# B&R Automation Studio project A2019059_Linka_Power_CP (part 62)

#### Main.st - Init, cyclic, exit code
```iecst
// ----------------------------------------------------------------------------------------
//	Function:	mappView explorer
//  Version:	1.00
//	Changed:	07.01.2020
// ----------------------------------------------------------------------------------------

PROGRAM _INIT
	// ----------------------------------------------------------------------------------------
	// Copy pre-configured devices into list
	brsmemcpy(ADR(EXPL.PAR[0].device_list), ADR(EXPL_DEVICE_LIST), SIZEOF(EXPL_DEVICE_LIST));
	brsmemcpy(ADR(EXPL.PAR[1].device_list), ADR(EXPL_DEVICE_LIST), SIZEOF(EXPL_DEVICE_LIST));
	brsstrcpy(ADR(EXPL.PAR[0].device_active), ADR(EXPL.PAR[0].device_list[0]));
	brsstrcpy(ADR(EXPL.PAR[1].device_active), ADR(EXPL.PAR[1].device_list[0]));

	// ----------------------------------------------------------------------------------------
	// Allocate memory for file upload and download
	AsMemPartCreate_0.enable	:= TRUE;
	AsMemPartCreate_0.len		:= EXPL_UPLOAD_DOWNLOAD_SIZE;
	AsMemPartCreate_0();
	IF AsMemPartCreate_0.status <> 0 THEN
		step := CreateError(ERR_MEM_ALLOC, side, step, 'file upload and download alloc failed', ADR(EXPL));
	ELSE
		AsMemPartAllocClear_0.enable	:= TRUE;
		AsMemPartAllocClear_0.ident		:= AsMemPartCreate_0.ident;
		AsMemPartAllocClear_0.len		:= EXPL_UPLOAD_DOWNLOAD_SIZE;
		AsMemPartAllocClear_0();
		IF AsMemPartCreate_0.status <> 0 THEN
			step := CreateError(ERR_MEM_ALLOC, side, step, 'file upload and download clear failed', ADR(EXPL));
		END_IF
	END_IF

	// ----------------------------------------------------------------------------------------
	// Generate HTML messages for web upload
	upload_response[0]	:= '<html><body><form action="/uploadA.html" name="form_upload" method="post" enctype="multipart/form-data" >
	<label for="file-upload" style="font-weight:bold;font-family: sans-serif;font-size:16px;padding:10px 10px;10px;10px;" class="custom-file-upload">Upload</label>
	<input type="file" id="file-upload" style="display:none;" onchange="form.submit()" name="file_selected" content-type="application/octet-stream" />
	</form><body></html> ';
	WebServiceUpload[0].pServiceName := ADR('uploadA.html');
	upload_response[1]	:= '<html><body><form action="/uploadB.html" name="form_upload" method="post" enctype="multipart/form-data" >
	<label for="file-upload" style="font-weight:bold;font-family: sans-serif;font-size:16px;padding:10px 10px;10px;10px;" class="custom-file-upload">Upload</label>
	<input type="file" id="file-upload" style="display:none;" onchange="form.submit()" name="file_selected" content-type="application/octet-stream" />
	</form><body></html> ';
	WebServiceUpload[1].pServiceName := ADR('uploadB.html');
END_PROGRAM

PROGRAM _CYCLIC
	// ----------------------------------------------------------------------------------------
	// Web service driver for file upload
	WebServiceUpload[side].enable 			:= TRUE;
	WebServiceUpload[side].option 			:= httpOPTION_HTTP_11 + httpOPTION_SERVICE_TYPE_NAME;
	WebServiceUpload[side].pRequestData  	:= AsMemPartAllocClear_0.mem;
	WebServiceUpload[side].requestDataSize 	:= EXPL_UPLOAD_DOWNLOAD_SIZE;
	WebServiceUpload[side].pResponseData 	:= ADR(upload_response[side]);
	WebServiceUpload[side].responseDataLen 	:= brsstrlen(ADR(upload_response[side]));
	WebServiceUpload[side]();

	// Reset send command
	IF(WebServiceUpload[side].send = TRUE)  THEN
		WebServiceUpload[side].send := FALSE;
	// Send response when page is loaded or data is posted
	ELSIF(WebServiceUpload[side].status = ERR_OK AND WebServiceUpload[side].send = FALSE) THEN
		WebServiceUpload[side].send := TRUE;
	// New upload data arrived
	ELSIF(WebServiceUpload[side].send = FALSE AND WebServiceUpload[side].requestDataLen > 0) THEN
		EXPL.CMD[side].upload := 1;
	END_IF

	// ------------------------------------------------------------------------------------------------
	// Set switches for HMI, these buttons are enabled if there is at least one file or directory
	IF(EXPL.DAT[side].item_num > 0) THEN
		EXPL.VIS[side].enable_button_set_1 := 1;
	ELSE
		EXPL.VIS[side].enable_button_set_1 := 0;
	END_IF

	// ------------------------------------------------------------------------------------------------
	// Generate device name list for drop down box
	brsmemset(ADR(EXPL.VIS[side].device_list), 0, SIZEOF(EXPL.VIS[side].device_list));
	FOR lx := 0 TO SIZEOF(EXPL.VIS[side].device_list)/SIZEOF(EXPL.VIS[side].device_list[0]) - 1 DO
		IF (EXPL.PAR[side].device_list[lx] <> '') THEN
			String2DataProvider(ADR(EXPL.PAR[side].device_list[lx]), ADR(EXPL.VIS[side].device_list[lx]));
		END_IF
	END_FOR;

	// ------------------------------------------------------------------------------------------------
	// Handle double click for directory change and file view
	IF(EXPL.VIS[side].double_click_event > 0) THEN
		double_click_timer.PT := 50;
		double_click_timer.IN := 1;
		double_click_timer();
		IF(EXPL.VIS[side].double_click_event > 1) THEN
			double_click_timer.IN := 0;
			double_click_timer();
			EXPL.VIS[side].double_click_event := 0;
			IF(brsmemcmp(ADR(EXPL.DAT[side].item_list[EXPL.VIS[side].item_selected]), ADR('(DIR)'), 5) = 0 OR EXPL.DAT[side].item_list[EXPL.VIS[side].item_selected] = '..') THEN
				EXPL.CMD[side].dir_change := 1;
			ELSE
				EXPL.CMD[side].view_file := 1;
			END_IF
		END_IF
	END_IF
	IF(double_click_timer.Q) THEN
		double_click_timer.IN := 0;
		double_click_timer();
		IF(EXPL.VIS[side].double_click_event > 0) THEN
			EXPL.VIS[side].double_click_event := EXPL.VIS[side].double_click_event - 1;
		END_IF
	END_IF

	//--------------------------------------------------------------------------------------------------
	// Check if parameters are valid
	IF (EXPL.PAR[side].device_active = '') THEN
		step := CreateError(ERR_DEVICE_UNDEFINED, side, step, 'device is not defined', ADR(EXPL));
		RETURN;
	END_IF
	IF (brsstrlen(ADR(EXPL.PAR[side].dir_path)) >= EXPL_DIR_PATH_LENGTH) THEN
		step := CreateError(ERR_PATH_CRITICAL, side, step, 'directory path critical error', ADR(EXPL));
		RETURN;
	END_IF

	// ------------------------------------------------------------------------------------------------
	// Track filter change
	IF (FILTER_AUTO_REFRESH AND brsstrcmp(ADR(old_filter[side]), ADR(EXPL.PAR[side].item_filter)) <> 0) THEN
		brsstrcpy(ADR(old_filter[side]), ADR(EXPL.PAR[side].item_filter));
		EXPL.CMD[side].refresh	:= 1;
	END_IF

	// ------------------------------------------------------------------------------------------------
	// Track device name change
	IF(device_active_old[side] <> EXPL.PAR[side].device_active) THEN
		EXPL.PAR[side].dir_path := '';
		EXPL.CMD[side].refresh	:= 1;
	END_IF
	device_active_old[side] := EXPL.PAR[side].device_active;

	// ------------------------------------------------------------------------------------------------
	// Stop here if no command is set
	IF (EXPL.CMD[side].refresh = 0 AND EXPL.CMD[side].dir_change = 0 AND EXPL.CMD[side].dir_create = 0 AND EXPL.CMD[side].copy = 0 AND EXPL.CMD[side].copy_all = 0 AND EXPL.CMD[side].delete = 0 AND EXPL.CMD[side].rename = 0 AND EXPL.CMD[side].view_file = 0 AND EXPL.CMD[side].download = 0 AND EXPL.CMD[side].upload = 0) THEN
		// --------------------------------------------------------------------------------------------
		// Show current state
		EXPL.status := 'Waiting...';
		// --------------------------------------------------------------------------------------------
		// If selection is out of range set it to maximum
		IF ((EXPL.VIS[side].item_selected > EXPL.DAT[side].item_num - 1) AND (EXPL.DAT[side].item_num <> 0)) THEN
			EXPL.VIS[side].item_selected := EXPL.DAT[side].item_num - 1;
		END_IF
		side := NOT side;
		// Enable buttons when command is active
		EXPL.VIS[0].enable_button_set_2 := 1;
		EXPL.VIS[1].enable_button_set_2 := 1;
		RETURN;
	END_IF

	// Disable buttons when command is active
	EXPL.VIS[0].enable_button_set_1 := 0;
	EXPL.VIS[1].enable_button_set_1 := 0;
	EXPL.VIS[0].enable_button_set_2 := 0;
	EXPL.VIS[1].enable_button_set_2 := 0;
	//**************************************************************************************************
	// Cyclic Part
	//**************************************************************************************************
	CASE step OF
		//**********************************************************************************************
		// Wait for command
		//**********************************************************************************************
		EXP_WAIT:
			// ----------------------------------------------------------------------------------------
			// Refresh direcrory information
			IF (EXPL.CMD[side].refresh = 1) THEN
				step := EXP_READ_DIR;
			END_IF
			// ----------------------------------------------------------------------------------------
			// Change active directory
			IF (EXPL.CMD[side].dir_change = 1) THEN
				// ------------------------------------------------------------------------------------
				// Check if directory name is empty
				IF (EXPL.DAT[side].item_list[EXPL.VIS[side].item_selected] = '') THEN
				step := CreateError(ERR_EMPTY_ITEM, side, step, 'directory name is empty', ADR(EXPL));
				// Check if directory name is valid
				ELSIF((brsmemcmp(ADR(EXPL.DAT[side].item_list[EXPL.VIS[side].item_selected]), ADR('(DIR)'), 5) <> 0) AND (EXPL.DAT[side].item_list[EXPL.VIS[side].item_selected] <> '..'))  THEN
					step := CreateError(ERR_INVALID_ITEM_NAME, side, step, 'this is not a valid directory name', ADR(EXPL));
				// Check if new directory name fits into string
				ELSIF(brsstrlen(ADR(EXPL.DAT[side].item_list[EXPL.VIS[side].item_selected])) - 5 + brsstrlen(ADR(EXPL.PAR[side].dir_path)) + 1 >= EXPL_DIR_PATH_LENGTH) THEN
					step := CreateError(ERR_PATH_EXCEEDS_MAX, side, step, 'directory path exceeds maximum length', ADR(EXPL));
				ELSE
					step := EXP_DIR_CHANGE;
				END_IF
			END_IF
			// ----------------------------------------------------------------------------------------
			// Create a new directory
			IF (EXPL.CMD[side].dir_create = 1) THEN
				// ------------------------------------------------------------------------------------
				// Check if new directory name is empty
				IF (EXPL.PAR[side].new_name = '') THEN
					step := CreateError(ERR_EMPTY_ITEM, side, step, 'directory name is empty', ADR(EXPL));
				// Check if new directory name fits into path string
				ELSIF(brsstrlen(ADR(EXPL.PAR[side].new_name)) + brsstrlen(ADR(EXPL.PAR[side].dir_path)) + 1 >= EXPL_DIR_PATH_LENGTH) THEN
					step := CreateError(ERR_PATH_EXCEEDS_MAX, side, step, 'directory path name exceeds maximum length', ADR(EXPL));
				// Check if new directory name fits into directory name string
				ELSIF(brsstrlen(ADR(EXPL.PAR[side].new_name)) + 5 >= EXPL_ITEM_LENGTH) THEN
					step := CreateError(ERR_DIR_EXCEEDS_MAX, side, step, 'directory name exceeds maximum length', ADR(EXPL));
				ELSE
					step := EXP_DIR_CREATE;
				END_IF
			END_IF
			// ----------------------------------------------------------------------------------------
			// Copy one file
			IF (EXPL.CMD[side].copy = 1) THEN
				// ------------------------------------------------------------------------------------
				// Make sure that user chooses a valid item
				IF (EXPL.DAT[side].item_list[EXPL.VIS[side].item_selected] = '..') THEN
					step := CreateError(ERR_INVALID_ITEM_NAME, side, step, 'this is not a valid item name', ADR(EXPL));
				ELSIF(brsmemcmp(ADR(EXPL.DAT[side].item_list[EXPL.VIS[side].item_selected]), ADR('(DIR)'), 5) = 0)	THEN
					step := EXP_DIR_COPY;
				ELSE
					step := EXP_FILE_COPY;
				END_IF
			END_IF
			// ----------------------------------------------------------------------------------------
			// Copy all files and folders in this directory
			IF (EXPL.CMD[side].copy_all = 1) THEN
				step := EXP_COPY_ALL;
			END_IF
			// ----------------------------------------------------------------------------------------
			// View selected file
			IF (EXPL.CMD[side].view_file = 1) THEN
				step := EXP_FILE_VIEW;
			END_IF
			// ----------------------------------------------------------------------------------------
			// Download selected file
			IF (EXPL.CMD[side].download = 1) THEN
				// Make sure download is not directory
				IF(brsmemcmp(ADR(EXPL.DAT[side].item_list[EXPL.VIS[side].item_selected]), ADR('(DIR)'), 5) <> 0) THEN
					EXPL.VIS[side].download_file_url := '';
					step := EXP_FILE_DOWNLOAD;
				ELSE
					step := CreateError(ERR_DIR_DOWNLOAD, side, step, 'downloading a directory is not supported', ADR(EXPL));
				END_IF
			END_IF
			// ----------------------------------------------------------------------------------------
			// Upload a new file
			IF (EXPL.CMD[side].upload = 1) THEN
				step := EXP_FILE_UPLOAD;
			END_IF
			// ----------------------------------------------------------------------------------------
			// Delete the selected file
			IF (EXPL.CMD[side].delete = 1) THEN
				// Check if directory name is empty
				IF (EXPL.DAT[side].item_list[EXPL.VIS[side].item_selected] = '')	THEN
					step := CreateError(ERR_EMPTY_ITEM, side, step, 'item name is empty', ADR(EXPL));
				// Check if new directory name fits into string
				ELSIF(brsstrlen(ADR(EXPL.DAT[side].item_list[EXPL.VIS[side].item_selected])) + brsstrlen(ADR(EXPL.PAR[side].dir_path)) + 1 >= EXPL_DIR_PATH_LENGTH + EXPL_ITEM_LENGTH) THEN
					step := CreateError(ERR_PATH_EXCEEDS_MAX, side, step, 'directory path exceeds maximum length', ADR(EXPL));
				// Make sure that a valid item was selected
				ELSIF(EXPL.DAT[side].item_list[EXPL.VIS[side].item_selected] = '..') THEN
					step := CreateError(ERR_INVALID_ITEM_NAME, side, step, 'this is not a valid item name', ADR(EXPL));
				// Delete a directory
				ELSIF(brsmemcmp(ADR(EXPL.DAT[side].item_list[EXPL.VIS[side].item_selected]), ADR('(DIR)'), 5) = 0)	THEN
					step := EXP_DIR_DELETE;
				// Delete a file
				ELSE
					step := EXP_FILE_DELETE;
				END_IF
			END_IF
			// ----------------------------------------------------------------------------------------
			// Rename file or directory
			IF (EXPL.CMD[side].rename = 1) THEN
				// ------------------------------------------------------------------------------------
				// Check if new directory name is empty
				IF (EXPL.PAR[side].new_name = '') THEN
					step := CreateError(ERR_EMPTY_ITEM, side, step, 'new name is empty', ADR(EXPL));
				// Make sure that a valid item was selected
				ELSIF (EXPL.DAT[side].item_list[EXPL.VIS[side].item_selected] = '..') THEN
					step := CreateError(ERR_INVALID_ITEM_NAME, side, step, 'this is not a valid item name', ADR(EXPL));
				// Rename a directory
				ELSIF(brsmemcmp(ADR(EXPL.DAT[side].item_list[EXPL.VIS[side].item_selected]), ADR('(DIR)'), 5) = 0)	THEN
					step := EXP_DIR_RENAME;
				// Rename a file
				ELSE
					step := EXP_FILE_RENAME;
				END_IF
			END_IF

			// Clear errors on new command
			brsmemset(ADR(EXPL.ERR), 0, SIZEOF(EXPL.ERR));

		//**********************************************************************************************
		// Read directory information
		//**********************************************************************************************
		EXP_READ_DIR:
			// Show current state
			animation := animation := WorkingStatus(ADR(EXPL), ADR('reading directory...'), animation);
			// ----------------------------------------------------------------------------------------
			// Clear all entrys
			brsmemset(ADR(EXPL.DAT[side]), 0, SIZEOF(EXPL.DAT[side]));
			EXPL.VIS[side].item_selected := 0;
			EXPL.DAT[side].item_num := 0;
			// ----------------------------------------------------------------------------------------
			// Add .. for directory up
			IF(EXPL.PAR[side].dir_path <> '/' AND EXPL.PAR[side].dir_path <> '') THEN
				EXPL.DAT[side].item_list[0] := '..';
				EXPL.DAT[side].item_num := 1;
			END_IF
			// ----------------------------------------------------------------------------------------
			// Set parameters and get device dir
			DInfo.enable 	:= 1;
			DInfo.pDevice	:= ADR(EXPL.PAR[side].device_active);
			DInfo.pPath 	:= ADR(EXPL.PAR[side].dir_path);
			DInfo();

			// ----------------------------------------------------------------------------------------
			// OK
			IF (DInfo.status = OK) THEN
				step := EXP_READ_DIR_1;
			// ----------------------------------------------------------------------------------------
			// Device is not available
			ELSIF (DInfo.status = fiERR_FILE_DEVICE) THEN
			 	EXPL.DAT[side].item_list[0] := 'not connected';
				step := CreateError(DInfo.status, side, step, 'not connected', ADR(EXPL));
			// ----------------------------------------------------------------------------------------
			// Device is not available
			ELSIF (DInfo.status = fiERR_DEVICE_MANAGER) THEN
				EXPL.DAT[side].item_list[0] := 'not connected';
				step := CreateError(DInfo.status, side, step, 'check device name and path', ADR(EXPL));
			// Error
			ELSIF (DInfo.status <> ERR_FUB_BUSY) THEN
				step := CreateError(DInfo.status, side, step, 'error dir info', ADR(EXPL));
			END_IF
		//**********************************************************************************************
		// Open directory
		//**********************************************************************************************
		EXP_READ_DIR_1:
			DOpen.enable 	:= 1;
			DOpen.pDevice	:= ADR(EXPL.PAR[side].device_active);
			DOpen.pName 	:= ADR(EXPL.PAR[side].dir_path);
			DOpen();

			// ----------------------------------------------------------------------------------------
			// OK
			IF (DOpen.status = OK) THEN
				has_oversized_items := FALSE;
				step := EXP_READ_DIR_2;
			// Error
			ELSIF (DOpen.status <> ERR_FUB_BUSY) THEN
				step := CreateError(DOpen.status, side, step, 'error dir open', ADR(EXPL));
			END_IF;
		//**********************************************************************************************
		// Read file directory information
		//**********************************************************************************************
	 	EXP_READ_DIR_2:
			DRead.enable 	:= 1;
			DRead.ident		:= DOpen.ident;
			DRead.pData 	:= ADR(lDirReadData);
			DRead.data_len 	:= SIZEOF(lDirReadData);
			DRead();

			// ----------------------------------------------------------------------------------------
			// OK
			IF (DRead.status = OK) THEN
				// ------------------------------------------------------------------------------------
				// Verify that we still have space in list
				IF (EXPL.DAT[side].item_num < SIZEOF(EXPL.DAT[side].item_list)/SIZEOF(EXPL.DAT[side].item_list[0])) THEN
					// --------------------------------------------------------------------------------
					// Make sure file name contains filter
					IF (brsstrlen(ADR(EXPL.PAR[side].item_filter)) = 0 OR IsInstr(ADR(lDirReadData.Filename), ADR(EXPL.PAR[side].item_filter))) THEN
						brsmemset(ADR(tmp_str1), 0, SIZEOF(tmp_str1));
						// ----------------------------------------------------------------------------
						// Read file information
						IF (lDirReadData.Mode = fiFILE) THEN
							IF (brsstrlen(ADR(lDirReadData.Filename)) < EXPL_ITEM_LENGTH) THEN
								brsstrcpy(ADR(tmp_str1), ADR(lDirReadData.Filename));
								// --------------------------------------------------------------------
								// Generate file size
								IF (lDirReadData.Filelength > 999999) THEN
									brsitoa(lDirReadData.Filelength/1000000, ADR(tmp_str2));
									brsstrcat(ADR(tmp_str2), ADR('M'));
								ELSIF (lDirReadData.Filelength > 999) THEN
									brsitoa(lDirReadData.Filelength/1000, ADR(tmp_str2));
									brsstrcat(ADR(tmp_str2), ADR('K'));
								ELSE
									brsitoa(lDirReadData.Filelength, ADR(tmp_str2));
								END_IF
								InsertRecName(ADR(EXPL), tmp_str1, tmp_str2, side);
								EXPL.DAT[side].item_num := EXPL.DAT[side].item_num + 1;
							ELSE
								has_oversized_items := TRUE;
							END_IF
						// ----------------------------------------------------------------------------
						// Read directory information
						ELSIF (brsstrcmp(ADR(lDirReadData.Filename), ADR('.')) <> 0 AND brsstrcmp(ADR(lDirReadData.Filename), ADR('..')) <> 0 AND brsstrcmp(ADR(lDirReadData.Filename), ADR('System Volume Information')) <> 0) THEN
							IF (brsstrlen(ADR(lDirReadData.Filename)) < EXPL_ITEM_LENGTH-5) THEN
								// Copy directory name
								tmp_str1 := '(DIR)';
								brsstrcat(ADR(tmp_str1), ADR(lDirReadData.Filename));
								InsertRecName(ADR(EXPL), tmp_str1, '', side);
								EXPL.DAT[side].item_num := EXPL.DAT[side].item_num + 1;
							ELSE
								has_oversized_items := TRUE;
							END_IF
						END_IF
					END_IF
				ELSE
					step := CreateError(ERR_MAX_FILES_REACHED, side, step, 'maximum number of files reached', ADR(EXPL));
				END_IF
			// Last entry reached
			ELSIF (DRead.status = fiERR_NO_MORE_ENTRIES) THEN
				step := EXP_READ_DIR_3;
			// Error
			ELSIF (DRead.status <> ERR_FUB_BUSY) THEN
				step := CreateError(DRead.status, side, step, 'error dir read', ADR(EXPL));
			END_IF
		//**********************************************************************************************
		// Close directory information
		//**********************************************************************************************
		EXP_READ_DIR_3:
			DClose.enable 	:= 1;
			DClose.ident	:= DOpen.ident;
			DClose();

			// ----------------------------------------------------------------------------------------
			// OK
			IF (DClose.status = OK) THEN
				// Select item after copy->refresh
				IF(do_select <> 0) THEN
					FOR ly:=0 TO EXPL.DAT[NOT USINT_TO_BOOL(do_select-1)].item_num DO
						IF(EXPL.DAT[USINT_TO_BOOL(do_select-1)].item_list[EXPL.VIS[USINT_TO_BOOL(do_select-1)].item_selected] = EXPL.DAT[NOT USINT_TO_BOOL(do_select-1)].item_list[ly]) THEN
							EXIT;
						END_IF
					END_FOR;
					EXPL.VIS[NOT USINT_TO_BOOL(do_select-1)].item_selected := ly;
					do_select := 0;
				END_IF
				// Reset command and return to wait state
				EXPL.CMD[side].refresh	:= 0;
				DClose.ident			:= 0;
				IF(has_oversized_items) THEN
					step := CreateError(ERR_NAME_EXCEEDS_MAX, side, step, 'one or more names exceeds maximum length', ADR(EXPL));
				ELSE
					step := EXP_WAIT;
				END_IF
			// Error
			ELSIF (DClose.status <> ERR_FUB_BUSY) THEN
				step := CreateError(DClose.status, side, step, 'error dir close', ADR(EXPL));
			END_IF
		//**********************************************************************************************
		// Change directory
		//**********************************************************************************************
		EXP_DIR_CHANGE:
			// ----------------------------------------------------------------------------------------
			// Move one directory up
			IF (EXPL.DAT[side].item_list[EXPL.VIS[side].item_selected] = '..') THEN
				lx := brsstrlen(ADR(EXPL.PAR[side].dir_path));
				WHILE lx>0 DO
					IF(brsmemcmp(ADR(EXPL.PAR[side].dir_path) + lx, ADR('/'), 1) = 0) THEN
						EXIT;
					ELSE
						brsmemset(ADR(EXPL.PAR[side].dir_path) + lx, 0, 1);
					END_IF
					lx := lx -1;
				END_WHILE
				brsmemset(ADR(EXPL.PAR[side].dir_path) + lx, 0, 1);
			// ----------------------------------------------------------------------------------------
			// Move one directory down
			ELSE
				brsstrcat(ADR(EXPL.PAR[side].dir_path), ADR('/'));
				brsstrcat(ADR(EXPL.PAR[side].dir_path), ADR(EXPL.DAT[side].item_list[EXPL.VIS[side].item_selected]) + 5);
				EXPL.CMD[side].refresh := 1;
			END_IF
			// Reset command and return to wait state
			EXPL.VIS[side].item_selected	:= 0;
			EXPL.CMD[side].dir_change 		:= 0;
			EXPL.CMD[side].refresh 			:= 1;
			step							:= EXP_WAIT;
		//**********************************************************************************************
		// Copy all items
		//**********************************************************************************************
		EXP_COPY_ALL:
			// Show current state
			animation := animation := WorkingStatus(ADR(EXPL), ADR('copying files and folders...'), animation);

			EXPL.VIS[side].item_selected := 0;
			// ----------------------------------------------------------------------------------------
			// Skip dots at the beginning of the list
			IF (EXPL.DAT[side].item_list[EXPL.VIS[side].item_selected] = '..') THEN
				EXPL.VIS[side].item_selected := EXPL.VIS[side].item_selected + 1;
			END_IF
			// Check first entry
			IF(brsmemcmp(ADR(EXPL.DAT[side].item_list[EXPL.VIS[side].item_selected]), ADR('(DIR)'), 5) = 0) THEN
				step := EXP_DIR_COPY;
			ELSE
				step := EXP_FILE_COPY;
			END_IF
		//**********************************************************************************************
		// Copy files
		//**********************************************************************************************
		EXP_FILE_COPY:
			// Show current state
			animation := WorkingStatus(ADR(EXPL), ADR('copying file...'), animation);

			// -----------------------------------------------------------------.----------------------
			// Proceed with copy all until last file is copied
			IF ((EXPL.VIS[side].item_selected < SIZEOF(EXPL.DAT[side].item_list)/SIZEOF(EXPL.DAT[side].item_list[0])) AND (EXPL.VIS[side].item_selected < EXPL.DAT[side].item_num)) THEN
				// ------------------------------------------------------------------------------------
				// Check if file name is empty
				IF (EXPL.DAT[side].item_list[EXPL.VIS[side].item_selected] <> '') THEN
					// --------------------------------------------------------------------------------
					// Check if new file name fits into string
					IF(brsstrlen(ADR(EXPL.DAT[side].item_list[EXPL.VIS[side].item_selected])) < EXPL_ITEM_LENGTH) THEN
						// ----------------------------------------------------------------------------
						// Initialize copy structure
						CreateCompletePath(EXPL.PAR[side].dir_path, EXPL.DAT[side].item_list[EXPL.VIS[side].item_selected], ADR(tmp_str3));
						CreateCompletePath(EXPL.PAR[NOT side].dir_path, EXPL.DAT[side].item_list[EXPL.VIS[side].item_selected], ADR(tmp_str4));
						FCopy.enable 	:= 1;
						FCopy.pSrcDev	:= ADR(EXPL.PAR[side].device_active);
						FCopy.pSrc		:= ADR(tmp_str3);
						FCopy.pDestDev  := ADR(EXPL.PAR[NOT side].device_active);
						FCopy.pDest		:= ADR(tmp_str4);
						FCopy.option 	:= FILE_OW_DETMEM;
						FCopy();

						// ----------------------------------------------------------------------------
						// OK
						IF (FCopy.status = OK AND EXPL.CMD[side].copy = 1) THEN
							// Select entry, reset command and refresh directory
							IF(COPY_AUTO_REFRESH = TRUE) THEN
								EXPL.CMD[NOT side].refresh := 1;
							END_IF
							IF(COPY_AUTO_SELECT = TRUE) THEN
								do_select := BOOL_TO_USINT(side) + 1;
							END_IF
							EXPL.CMD[side].copy	:= 0;
							step := EXP_WAIT;
						// ----------------------------------------------------------------------------
						// Proceed with next file
						ELSIF (FCopy.status = OK) THEN
							EXPL.VIS[side].item_selected := EXPL.VIS[side].item_selected + 1;
						ELSIF (FCopy.status <> ERR_FUB_BUSY) THEN
							step := CreateError(FCopy.status, side, step, 'error copying file', ADR(EXPL));
						END_IF
					// File name is too long
					ELSE
						step := CreateError(ERR_NAME_EXCEEDS_MAX, side, step, 'file name exceeds maximum length', ADR(EXPL));
					END_IF
				// File name  is empty
				ELSE
					step := CreateError(ERR_EMPTY_ITEM, side, step, 'file name is empty', ADR(EXPL));
				END_IF
			// ----------------------------------------------------------------------------------------
			// Finish copy all
			ELSE
				// Reset command and refresh directory
				IF(COPY_AUTO_REFRESH = TRUE) THEN
					EXPL.CMD[NOT side].refresh := 1;
				END_IF
				EXPL.CMD[side].copy_all			:= 0;
				EXPL.VIS[side].item_selected 	:= 0;
				step							:= EXP_WAIT;
			END_IF
		//**********************************************************************************************
		// Copy directory
		//**********************************************************************************************
		EXP_DIR_COPY:
			// Show current state
			animation := WorkingStatus(ADR(EXPL), ADR('copying directory...'), animation);

			// ----------------------------------------------------------------------------------------
			// Proceed with copy all until last file is copied
			IF ((EXPL.VIS[side].item_selected < SIZEOF(EXPL.DAT[side].item_list)/SIZEOF(EXPL.DAT[side].item_list[0])) AND (EXPL.VIS[side].item_selected < EXPL.DAT[side].item_num)) THEN
				IF (EXPL.DAT[side].item_list[EXPL.VIS[side].item_selected] <> '') THEN
					// --------------------------------------------------------------------------------
					// Check if new directory name fits into path string
					IF(brsstrlen(ADR(EXPL.DAT[side].item_list[EXPL.VIS[side].item_selected])) + brsstrlen(ADR(EXPL.PAR[NOT side].dir_path)) + 1 < EXPL_DIR_PATH_LENGTH) THEN
						// ----------------------------------------------------------------------------
						// Initialize copy structure
						CreateCompletePath(EXPL.PAR[side].dir_path, EXPL.DAT[side].item_list[EXPL.VIS[side].item_selected], ADR(tmp_str3));
						CreateCompletePath(EXPL.PAR[NOT side].dir_path, EXPL.DAT[side].item_list[EXPL.VIS[side].item_selected], ADR(tmp_str4));
						DCopy.enable 	:= 1;
						DCopy.pSrcDev	:= ADR(EXPL.PAR[side].device_active);
						DCopy.pSrcDir	:= ADR(tmp_str3);
						DCopy.pDestDev 	:= ADR(EXPL.PAR[NOT side].device_active);
						DCopy.pDestDir 	:= ADR(tmp_str4);
						DCopy.option 	:= fiOVERWRITE;
						DCopy();

						// ----------------------------------------------------------------------------
						// OK
						IF (DCopy.status = OK AND EXPL.CMD[side].copy = 1) THEN
							// Reset command and refresh directory
							IF(COPY_AUTO_REFRESH = TRUE) THEN
								EXPL.CMD[NOT side].refresh := 1;
							END_IF
							IF (COPY_AUTO_SELECT = TRUE) THEN
								do_select := BOOL_TO_USINT(side) + 1;
							END_IF
							EXPL.CMD[side].copy	:= 0;
							step := EXP_WAIT;
						// ----------------------------------------------------------------------------
						// Proceed with next directory
						ELSIF (DCopy.status = OK) THEN
							EXPL.VIS[side].item_selected := EXPL.VIS[side].item_selected + 1;
							// Switch to file copy when no more directory can be found
							IF(brsmemcmp(ADR(EXPL.DAT[side].item_list[EXPL.VIS[side].item_selected]), ADR('(DIR)'), 5) <> 0) THEN
								step := EXP_FILE_COPY;
							END_IF
						END_IF
					// Error
					ELSIF (DCopy.status <> ERR_FUB_BUSY) THEN
						step := CreateError(DCopy.status, side, step, 'error copying directory', ADR(EXPL));
					// Directory name is too long
					ELSE
						step := CreateError(ERR_PATH_EXCEEDS_MAX, side, step, 'directory path name exceeds maximum length', ADR(EXPL));
					END_IF
				// Directory name is empty
				ELSE
					step := CreateError(ERR_EMPTY_ITEM, side, step, 'directory name is empty', ADR(EXPL));
				END_IF
			// ----------------------------------------------------------------------------------------
			// Finish copy all
			ELSE
				// Reset command and refresh directory
				IF (COPY_AUTO_REFRESH = TRUE) THEN
					EXPL.CMD[NOT side].refresh := 1;
				END_IF
				EXPL.CMD[side].copy_all := 0;
				EXPL.VIS[side].item_selected := 0;
				step := EXP_WAIT;
			END_IF
		//**********************************************************************************************
		// Delete selected file
		//**********************************************************************************************
		EXP_FILE_DELETE:
			// Show current state
			animation := WorkingStatus(ADR(EXPL), ADR('deleting file...'), animation);

			// ----------------------------------------------------------------------------------------
			// Initialize file delete structure
			CreateCompletePath(EXPL.PAR[side].dir_path, EXPL.DAT[side].item_list[EXPL.VIS[side].item_selected], ADR(tmp_str3));
			FDelete.enable		:= 1;
			FDelete.pDevice 	:= ADR(EXPL.PAR[side].device_active);
			FDelete.pName		:= ADR(tmp_str3);
			FDelete();

			// ----------------------------------------------------------------------------------------
			// OK
			IF (FDelete.status = OK) THEN
				// Reset command and return to wait state
				EXPL.CMD[side].delete 	:= 0;
				EXPL.CMD[side].refresh  := 1;
				step := EXP_WAIT;
			// Error
			ELSIF (FDelete.status <> ERR_FUB_BUSY) THEN
				step := CreateError(FDelete.status, side, step, 'error deleting file', ADR(EXPL));
			END_IF
		//**********************************************************************************************
		// Rename selected file
		//**********************************************************************************************
		EXP_FILE_RENAME:
			// Show current state
			animation := WorkingStatus(ADR(EXPL), ADR('renaming file...'), animation);

			// ----------------------------------------------------------------------------------------
			// Initialize file delete structure
			CreateCompletePath(EXPL.PAR[side].dir_path, EXPL.DAT[side].item_list[EXPL.VIS[side].item_selected], ADR(tmp_str2));
			CreateCompletePath(EXPL.PAR[side].dir_path, EXPL.PAR[side].new_name, ADR(tmp_str3));
			FRename.enable		:= 1;
			FRename.pDevice 	:= ADR(EXPL.PAR[side].device_active);
			FRename.pName		:= ADR(tmp_str2);
			FRename.pNewName	:= ADR(tmp_str3);
			FRename();

			// ----------------------------------------------------------------------------------------
			// OK
			IF (FRename.status = OK) THEN
				// Reset command and return to wait state
				EXPL.CMD[side].rename 	:= 0;
				EXPL.CMD[side].refresh  := 1;
				step := EXP_WAIT;
				// Error
			ELSIF (FRename.status <> ERR_FUB_BUSY) THEN
				step := CreateError(FRename.status, side, step, 'error renaming file', ADR(EXPL));
			END_IF
		//**********************************************************************************************
		// View selected file
		//**********************************************************************************************
		EXP_FILE_VIEW:
			CreateCompletePath(EXPL.PAR[side].dir_path, EXPL.DAT[side].item_list[EXPL.VIS[side].item_selected], ADR(tmp_str1));

			FOR lx:=0 TO SIZEOF(EXPL_VIEW_FILTER)/SIZEOF(EXPL_VIEW_FILTER[0]) - 1 DO
				IF(brsstrlen(ADR(tmp_str1)) >= brsstrlen(ADR(EXPL_VIEW_FILTER[lx])) AND EXPL_VIEW_FILTER[lx] <> '') THEN
					// --------------------------------------------------------------------------------
					// Verify that file name contains filter
					IF(brsmemcmp(ADR(tmp_str1) + brsstrlen(ADR(tmp_str1)) - brsstrlen(ADR(EXPL_VIEW_FILTER[lx])) , ADR(EXPL_VIEW_FILTER[lx]), brsstrlen(ADR(EXPL_VIEW_FILTER[lx]))) = 0) THEN
						EXPL.VIS[side].view_file_path := '/FileDevice:';
						brsstrcat(ADR(EXPL.VIS[side].view_file_path), ADR(EXPL.PAR[side].device_active));
						brsstrcat(ADR(EXPL.VIS[side].view_file_path), ADR(tmp_str1));
						EXPL.CMD[side].view_file := FALSE;
						EXPL.VIS[side].view_file := TRUE;
						step := EXP_WAIT;
						RETURN;
					END_IF
				END_IF
			END_FOR;
			step := CreateError(FRename.status, side, step, 'error this file extension is not supported for viewing', ADR(EXPL));
		//**********************************************************************************************
		// Download file
		//**********************************************************************************************
		EXP_FILE_DOWNLOAD:
			// ----------------------------------------------------------------------------------------
			// Initialize file open structure
			CreateCompletePath(EXPL.PAR[side].dir_path, EXPL.DAT[side].item_list[EXPL.VIS[side].item_selected], ADR(tmp_str1));
			FOpen.enable	:= TRUE;
			FOpen.pDevice 	:= ADR(EXPL.PAR[side].device_active);
			FOpen.pFile		:= ADR(tmp_str1);
			FOpen();

			// ----------------------------------------------------------------------------------------
			// OK
			IF (FOpen.status = OK) THEN
				// Make sure file fits into memory
				IF(FOpen.filelen <= EXPL_UPLOAD_DOWNLOAD_SIZE) THEN
					// Clear memory and reset web service
					brsmemset(AsMemPartAllocClear_0.mem, 0, EXPL_UPLOAD_DOWNLOAD_SIZE);
					WebserviceDownload.enable := FALSE;
					WebserviceDownload();
					step := EXP_FILE_DOWNLOAD_1;
				// File is too large
				ELSE
					tmp_str1 := 'download file exceeds maximum buffer size of ';
					brsitoa(EXPL_UPLOAD_DOWNLOAD_SIZE, ADR(tmp_str2));
					brsstrcat(ADR(tmp_str1), ADR(tmp_str2));
					brsstrcat(ADR(tmp_str1), ADR(' bytes'));
					step := CreateError(ERR_MEM_DOWNLOAD, side, step, tmp_str1, ADR(EXPL));
				END_IF;
			// Error
			ELSIF (FOpen.status <> ERR_FUB_BUSY) THEN
				step := CreateError(FOpen.status, side, step, 'error opening file for download', ADR(EXPL));
			END_IF
		//**********************************************************************************************
		// Download file
		//**********************************************************************************************
		EXP_FILE_DOWNLOAD_1:
			// ----------------------------------------------------------------------------------------
			// Initialize file read structure
			FRead.enable	:= TRUE;
			FRead.ident		:= FOpen.ident;
			FRead.len		:= FOpen.filelen;
			FRead.pDest		:= AsMemPartAllocClear_0.mem;
			FRead();

			// ----------------------------------------------------------------------------------------
			// OK
			IF (FRead.status = OK) THEN
				step := EXP_FILE_DOWNLOAD_2;
			// Error
			ELSIF (FRead.status <> ERR_FUB_BUSY) THEN
				step := CreateError(FRead.status, side, step, 'error reading file for download', ADR(EXPL));
			END_IF
		//**********************************************************************************************
		// Download file
		//**********************************************************************************************
		EXP_FILE_DOWNLOAD_2:
			// ----------------------------------------------------------------------------------------
			// Initialize file close structure
			FClose.enable	:= TRUE;
			FClose.ident	:= FOpen.ident;
			FClose();

			// ----------------------------------------------------------------------------------------
			// OK
			IF (FClose.status = OK) THEN
				download_timeout.IN := 0;
				download_timeout();
				step := EXP_FILE_DOWNLOAD_3;
			// Error
			ELSIF (FClose.status <> ERR_FUB_BUSY) THEN
				step := CreateError(FClose.status, side, step, 'error closing file for download', ADR(EXPL));
			END_IF
		//**********************************************************************************************
		// Download file - web service
		//**********************************************************************************************
		EXP_FILE_DOWNLOAD_3:
			// ----------------------------------------------------------------------------------------
			// Create response header
			response_header_data :=  'Content-Type: application/octet-stream; Content-Transfer-Encoding: binary; Content-Disposition: attachment; filename="';
			brsstrcpy(ADR(tmp_str1), ADR(EXPL.DAT[side].item_list[EXPL.VIS[side].item_selected]));
			ReplaceString(ADR(tmp_str1), ADR(' '), ADR('%20'));
			brsstrcat(ADR(response_header_data), ADR(tmp_str1));
			brsstrcat(ADR(response_header_data), ADR('"'));

			// ----------------------------------------------------------------------------------------
			// Pre-configure web service for download
			response_header.rawHeader.pData 	:= ADR(response_header_data);
			response_header.rawHeader.dataSize 	:= SIZEOF(response_header_data);
			response_header.rawHeader.dataLen 	:= brsstrlen(ADR(response_header_data));

			// ----------------------------------------------------------------------------------------
			// Start web service
			WebserviceDownload.enable 			:= TRUE;
			WebserviceDownload.option 			:= httpOPTION_HTTP_10 + httpOPTION_SERVICE_TYPE_NAME;
			WebserviceDownload.pResponseData 	:= AsMemPartAllocClear_0.mem;
			WebserviceDownload.pResponseHeader	:= ADR(response_header);
			WebserviceDownload.pServiceName 	:= ADR(tmp_str1);
			WebserviceDownload.responseDataLen 	:= FOpen.filelen;
			WebserviceDownload();

			// ----------------------------------------------------------------------------------------
			// Timeout if file is not pulled from browser
			download_timeout.IN := 1;
			download_timeout.PT := 300;
			download_timeout();
			IF(download_timeout.Q) THEN
				step := CreateError(ERR_TIMEOUT_DOWNLOAD, side, step, 'error download response timed out', ADR(EXPL));
			END_IF

			// ----------------------------------------------------------------------------------------
			// Set URL
			IF (WebserviceDownload.status = ERR_FUB_BUSY AND EXPL.VIS[side].download_file_url = '') THEN
				brsstrcat(ADR(EXPL.VIS[side].download_file_url), ADR(EXPL.DAT[side].item_list[EXPL.VIS[side].item_selected]));
			// Start sending data
			ELSIF (WebserviceDownload.status = OK AND WebserviceDownload.send = FALSE AND EXPL.VIS[side].download_file_url <> '') THEN
				WebserviceDownload.send := TRUE;
			// Sending data finished
			ELSIF (WebserviceDownload.send = TRUE) THEN
				WebserviceDownload.send := FALSE;
				step := EXP_FILE_DOWNLOAD_4;
			// Error
			ELSIF (WebserviceDownload.status <> ERR_FUB_BUSY AND WebserviceDownload.status <> OK) THEN
				step := CreateError(WebserviceDownload.status, side, step, 'error sending web response', ADR(EXPL));
			END_IF
		//**********************************************************************************************
		// Download file - web service
		//**********************************************************************************************
		EXP_FILE_DOWNLOAD_4:
			WebserviceDownload();

			// ----------------------------------------------------------------------------------------
			// Start sending data
			IF (WebserviceDownload.status = OK AND WebserviceDownload.send = FALSE) THEN
				WebserviceDownload.send := TRUE;
			// Sending data finished
			ELSIF (WebserviceDownload.send = TRUE) THEN
				WebserviceDownload.send := FALSE;
				EXPL.CMD[side].download	:= 0;
				step := EXP_WAIT;
			// Error
			ELSIF (WebserviceDownload.status <> ERR_FUB_BUSY) THEN
				step := CreateError(WebserviceDownload.status, side, step, 'error sending web response', ADR(EXPL));
			END_IF

		//**********************************************************************************************
		// Upload file - verify parameters
		//**********************************************************************************************
		EXP_FILE_UPLOAD:
			// Show current state
			animation := WorkingStatus(ADR(EXPL), ADR('uploading file...'), animation);

			// Make sure data fits into memory
			IF(WebServiceUpload[side].requestDataLen < EXPL_UPLOAD_DOWNLOAD_SIZE) THEN
				// Find file name start
				file_name_start := FindInMem(AsMemPartAllocClear_0.mem, WebServiceUpload[side].requestDataLen, ADR('filename="'), brsstrlen(ADR('filename="'))) + brsstrlen(ADR('filename="'));
				IF(file_name_start > 0) THEN
					// Find end of file name
					file_name_len := FindInMem(AsMemPartAllocClear_0.mem+file_name_start, WebServiceUpload[side].requestDataLen-file_name_start, ADR('"$r$n'), brsstrlen(ADR('"$r$n')));
					IF(file_name_len > 0) THEN
						// Make sure file name is not too long
						IF(file_name_len <= SIZEOF(file_name)) THEN
							// Store file name
							brsmemset(ADR(file_name), 0, SIZEOF(file_name));
							brsmemcpy(ADR(file_name), AsMemPartAllocClear_0.mem+file_name_start, file_name_len);
							// Find start of data
							file_data_start := FindInMem(AsMemPartAllocClear_0.mem, WebServiceUpload[side].requestDataLen, ADR('Content-Type:'), brsstrlen(ADR('Content-Type:'))) + brsstrlen(ADR('Content-Type:'));
							IF(file_data_start > 0) THEN
								// Find end of data
								file_data_start := FindInMem(AsMemPartAllocClear_0.mem+file_data_start, WebServiceUpload[side].requestDataLen-file_data_start, ADR('$r$n$r$n'), brsstrlen(ADR('$r$n$r$n'))) + brsstrlen(ADR('$r$n$r$n'))+file_data_start;
								file_data_len := FindInMem(AsMemPartAllocClear_0.mem+file_data_start, WebServiceUpload[side].requestDataLen-file_data_start, ADR('$r$n------'), brsstrlen(ADR('$r$n------')));
								// When file name and data is correct procceed with saving data to file
								IF(file_data_len > 0) THEN
									step := EXP_FILE_UPLOAD_1;
									RETURN;
								ELSE
									step := CreateError(ERR_SIZE_DATA_UPLOAD, side, step, 'data end not found in upload response', ADR(EXPL));
								END_IF
							// Data start not found in upload response
							ELSE
								step := CreateError(ERR_POS_DATA_UPLOAD, side, step, 'data start not found in upload response', ADR(EXPL));
							END_IF
						// File name is too long in upload response
						ELSE
							step := CreateError(ERR_LEN_NAME_UPLOAD, side, step, 'file name is too long in upload response', ADR(EXPL));
						END_IF
					// File name end not found in upload response
					ELSE
						step := CreateError(ERR_SIZE_NAME_UPLOAD, side, step, 'file name end not found in upload response', ADR(EXPL));
					END_IF
				// File name start not found in upload response
				ELSE
					step := CreateError(ERR_POS_NAME_UPLOAD, side, step, 'file name position not found in upload response', ADR(EXPL));
				END_IF
			// Upload file exceeds maximum buffer size
			ELSE
				tmp_str1 := 'upload file exceeds maximum buffer size of ';
				brsitoa(EXPL_UPLOAD_DOWNLOAD_SIZE, ADR(tmp_str2));
				brsstrcat(ADR(tmp_str1), ADR(tmp_str2));
				brsstrcat(ADR(tmp_str1), ADR(' bytes'));
				step := CreateError(ERR_MEM_UPLOAD, side, step, tmp_str1, ADR(EXPL));
			END_IF
			// Reset upload buffer and function block
			brsmemset(AsMemPartAllocClear_0.mem, 0, EXPL_UPLOAD_DOWNLOAD_SIZE);
			EXPL.VIS[side].reload_upload := TRUE;
			WebServiceUpload[side].enable := FALSE;
			WebServiceUpload[side]();
		//**********************************************************************************************
		// Upload file
		//**********************************************************************************************
		EXP_FILE_UPLOAD_1:
			// ----------------------------------------------------------------------------------------
			// Initialize file create structure
			CreateCompletePath(EXPL.PAR[side].dir_path, file_name, ADR(tmp_str1));
			FCreate.enable	:= TRUE;
			FCreate.pDevice := ADR(EXPL.PAR[side].device_active);
			FCreate.pFile	:= ADR(tmp_str1);
			FCreate();

			// ----------------------------------------------------------------------------------------
			// OK
			IF (FCreate.status = OK) THEN
				step := EXP_FILE_UPLOAD_2;
			// Error
			ELSIF (FCreate.status <> ERR_FUB_BUSY) THEN
				step := CreateError(FCreate.status, side, step, 'error creating file from upload', ADR(EXPL));
				// Reset upload buffer and function block
				brsmemset(AsMemPartAllocClear_0.mem, 0, EXPL_UPLOAD_DOWNLOAD_SIZE);
				EXPL.VIS[side].reload_upload := TRUE;
				WebServiceUpload[side].enable := FALSE;
				WebServiceUpload[side]();
				FCreate.enable	:= FALSE;
				FCreate();
			END_IF
		//**********************************************************************************************
		// Upload file
		//**********************************************************************************************
		EXP_FILE_UPLOAD_2:
			// Show current state
			animation := WorkingStatus(ADR(EXPL), ADR('upload - saving file...'), animation);

			// ----------------------------------------------------------------------------------------
			// Initialize file write structure
			FWrite.enable	:= TRUE;
			FWrite.ident	:= FCreate.ident;
			FWrite.len		:= file_data_len;
			FWrite.pSrc		:= AsMemPartAllocClear_0.mem + file_data_start;
			FWrite();

			// ----------------------------------------------------------------------------------------
			// OK
			IF (FWrite.status = OK) THEN
				step := EXP_FILE_UPLOAD_3;
			// Error
			ELSIF (FWrite.status <> ERR_FUB_BUSY) THEN
				step := CreateError(FWrite.status, side, step, 'error writing file from upload', ADR(EXPL));
			END_IF
		//**********************************************************************************************
		// Upload file
		//**********************************************************************************************
		EXP_FILE_UPLOAD_3:
			// ----------------------------------------------------------------------------------------
			// Initialize file close structure
			FClose.enable	:= TRUE;
			FClose.ident	:= FCreate.ident;
			FClose();

			// ----------------------------------------------------------------------------------------
			// OK
			IF (FClose.status = OK) THEN
				brsmemset(AsMemPartAllocClear_0.mem, 0, EXPL_UPLOAD_DOWNLOAD_SIZE);
				WebServiceUpload[side].enable := FALSE;
				WebServiceUpload[side]();
				EXPL.CMD[side].upload := 0;
				EXPL.CMD[side].refresh := 1;
				EXPL.VIS[side].reload_upload := TRUE;
				step := EXP_WAIT;
			// Error
			ELSIF (FClose.status <> ERR_FUB_BUSY) THEN
				step := CreateError(FClose.status, side, step, 'error closing file from upload', ADR(EXPL));
			END_IF
		//**********************************************************************************************
		// Create new directory
		//**********************************************************************************************
		EXP_DIR_CREATE:
			// Show current state
			animation := WorkingStatus(ADR(EXPL), ADR('creating directory...'), animation);

			// ----------------------------------------------------------------------------------------
			// Initialize directory create structure
			CreateCompletePath(EXPL.PAR[side].dir_path, EXPL.PAR[side].new_name, ADR(tmp_str3));
			DCreate.enable	:= 1;
			DCreate.pDevice := ADR(EXPL.PAR[side].device_active);
			DCreate.pName 	:= ADR(tmp_str3);
			DCreate();

			// ----------------------------------------------------------------------------------------
			// OK
			IF (DCreate.status = OK) THEN
				// Reset command and return to wait state
				EXPL.CMD[side].dir_create 	:= 0;
				EXPL.CMD[side].refresh 		:= 1;
				step := EXP_WAIT;
			// Error
			ELSIF (DCreate.status <> ERR_FUB_BUSY) THEN
				step := CreateError(DCreate.status, side, step, 'error creating directory', ADR(EXPL));
			END_IF
		//**********************************************************************************************
		// Delete selected directory
		//**********************************************************************************************
		EXP_DIR_DELETE:
			// Show current state
			animation := WorkingStatus(ADR(EXPL), ADR('deleting directory...'), animation);

			// ----------------------------------------------------------------------------------------
			// Initialize directory delete structure
			CreateCompletePath(EXPL.PAR[side].dir_path, EXPL.DAT[side].item_list[EXPL.VIS[side].item_selected], ADR(tmp_str3));
			DDelete.enable	:= 1;
			DDelete.pDevice := ADR(EXPL.PAR[side].device_active);
			DDelete.pName 	:= ADR(tmp_str3);
			DDelete();

			// ----------------------------------------------------------------------------------------
			// OK
			IF (DDelete.status = OK) THEN
				// Reset command and return to wait state
				EXPL.CMD[side].delete := 0;
				EXPL.CMD[side].refresh := 1;
				step := EXP_WAIT;
			// Error
			ELSIF (DDelete.status <> ERR_FUB_BUSY) THEN
				step := CreateError(DDelete.status, side, step, 'error deleting directory', ADR(EXPL));
			END_IF
		//**********************************************************************************************
		// Rename selected directory
		//**********************************************************************************************
		EXP_DIR_RENAME:
			// Show current state
			animation := WorkingStatus(ADR(EXPL), ADR('renaming directory...'), animation);

			// ----------------------------------------------------------------------------------------
			// Initialize file delete structure
			CreateCompletePath(EXPL.PAR[side].dir_path, EXPL.DAT[side].item_list[EXPL.VIS[side].item_selected], ADR(tmp_str2));
			CreateCompletePath(EXPL.PAR[side].dir_path, EXPL.PAR[side].new_name, ADR(tmp_str3));
			DRename.enable		:= 1;
			DRename.pDevice 	:= ADR(EXPL.PAR[side].device_active);
			DRename.pName		:= ADR(tmp_str2);
			DRename.pNewName	:= ADR(tmp_str3);
			DRename();

			// ----------------------------------------------------------------------------------------
			// OK
			IF (DRename.status = OK) THEN
				// Reset command and return to wait state
				EXPL.CMD[side].rename 	:= 0;
				EXPL.CMD[side].refresh  := 1;
				step := EXP_WAIT;
				// Error
			ELSIF (DRename.status <> ERR_FUB_BUSY) THEN
				step := CreateError(DRename.status, side, step, 'error renaming directory', ADR(EXPL));
			END_IF
	END_CASE

END_PROGRAM
```

#### Variables.var - Local variables
```iecst
(*Local constants*)
VAR CONSTANT
	OK : USINT := 0; (* CONSTANT for status OK *)
	FILTER_AUTO_REFRESH : BOOL := TRUE; (* Auto refresh when filter changes *)
	COPY_AUTO_SELECT : USINT := 1; (* Select target item after copying *)
	COPY_AUTO_REFRESH : USINT := 1; (* Refresh items after copying *)
END_VAR
(*Local Variables*)
VAR
	side : BOOL := FALSE; (* Current side *)
	step : expSTATE := (0); (* Main step index *)
	animation : USINT := 0; (* Animation for working status	*)
	do_select : USINT := 0; (* Select item after copying *)
	old_filter : ARRAY[0..1] OF STRING[EXPL_ITEM_LENGTH]; (* Track filter change *)
	has_oversized_items : BOOL;
	tmp_str1 : STRING[EXPL_DIR_PATH_LENGTH]; (* Temporary STRING variable *)
	tmp_str2 : STRING[EXPL_DIR_PATH_LENGTH]; (* Temporary STRING variable *)
	tmp_str3 : STRING[EXPL_DIR_PATH_LENGTH]; (* Temporary STRING variable *)
	tmp_str4 : STRING[EXPL_DIR_PATH_LENGTH]; (* Temporary STRING variable *)
	lx : UDINT := 0; (* Index	*)
	ly : UINT;
	double_click_timer : TON_10ms;
	device_active_old : ARRAY[0..1] OF STRING[40];
	response_header : httpResponseHeader_t;
	response_header_data : STRING[300];
	download_timeout : TON_10ms;
	upload_response : ARRAY[0..1] OF STRING[600];
	file_name_start : UDINT;
	file_name_len : UDINT;
	file_data_start : UDINT;
	file_data_len : UDINT;
	file_name : STRING[100];
END_VAR
(*Local function calls*)
VAR
	DInfo : DirInfo;
	DOpen : DirOpen;
	DRead : DirReadEx;
	DClose : DirClose;
	FWrite : FileWrite;
	FCreate : FileCreate;
	FOpen : FileOpen;
	FRead : FileReadEx;
	FClose : FileClose;
	FCopy : FileCopy;
	FDelete : FileDelete;
	FRename : FileRename;
	DCopy : DirCopy;
	DCreate : DirCreate;
	DDelete : DirDeleteEx;
	DRename : DirRename;
	lDirReadData : fiDIR_READ_EX_DATA;
	AsMemPartCreate_0 : AsMemPartCreate;
	AsMemPartAllocClear_0 : AsMemPartAllocClear;
	WebServiceUpload : ARRAY[0..1] OF httpService := [2((0))];
	WebserviceDownload : httpService := (0);
END_VAR
(*Local constants*)
VAR
	ERR_EMPTY_ITEM : UINT := 50000; (*Selected item name is empty	*)
	ERR_INVALID_ITEM_NAME : UINT := 50001; (*This is not a valid item name*)
	ERR_DEVICE_UNDEFINED : UINT := 50010; (*Device is not defined*)
	ERR_MAX_FILES_REACHED : UINT := 50100; (*Maximum number of files reached*)
	ERR_NAME_EXCEEDS_MAX : UINT := 50200; (*File name exceeds maximum length*)
	ERR_DIR_EXCEEDS_MAX : UINT := 50201; (*Directory name exceeds maximum length*)
	ERR_PATH_EXCEEDS_MAX : UINT := 50202; (*Directory path exceeds maximum length*)
	ERR_PATH_CRITICAL : UINT := 50203; (*Directory path critical error*)
	ERR_MEM_ALLOC : UINT := 50300; (*Memory allocation for file upload and download failed*)
	ERR_MEM_DOWNLOAD : UINT := 50310; (*Size of download file exceeds maximum*)
	ERR_TIMEOUT_DOWNLOAD : UINT := 50320; (*Download response timed out*)
	ERR_DIR_DOWNLOAD : UINT := 50330; (*Directories can not be downloaded*)
	ERR_POS_NAME_UPLOAD : UINT := 50400; (*Can not find filename in upload response*)
	ERR_SIZE_NAME_UPLOAD : UINT := 50401; (*Can not determine end of filename in upload response*)
	ERR_LEN_NAME_UPLOAD : UINT := 50402; (*Filename is too long in upload response*)
	ERR_POS_DATA_UPLOAD : UINT := 50403; (*Can not find data in upload response*)
	ERR_SIZE_DATA_UPLOAD : UINT := 50404; (*Can not determine end of data in upload response*)
	ERR_MEM_UPLOAD : UINT := 50410; (*Size of upload file exceeds maximum size*)
END_VAR
```

#### LocalFunctions.fun
```iecst
FUNCTION ReplaceString : BOOL
	VAR_INPUT
		dataSTR : UDINT;
		searchSTR : UDINT;
		replaceSTR : UDINT;
	END_VAR
	VAR
		idx : UDINT;
	END_VAR
END_FUNCTION

FUNCTION IsInstr : BOOL
	VAR_INPUT
		string1 : UDINT;
		string2 : UDINT;
	END_VAR
	VAR
		idx : UDINT;
	END_VAR
END_FUNCTION

FUNCTION FindInMem : UDINT
	VAR_INPUT
		data1 : UDINT;
		len1 : UDINT;
		data2 : UDINT;
		len2 : UDINT;
	END_VAR
	VAR
		idx : UDINT;
	END_VAR
END_FUNCTION

{REDUND_ERROR} FUNCTION CreateError : expSTATE (*TODO: Add your comment here*) (*$GROUP=User,$CAT=User,$GROUPICON=User.png,$CATICON=User.png*)
	VAR_INPUT
		nr : UINT;
		side : BOOL;
		step : expSTATE;
		text : STRING[150];
		EXPL : REFERENCE TO expMAIN;
	END_VAR
END_FUNCTION

FUNCTION InsertRecName : BOOL
	VAR_INPUT
		EXPL : REFERENCE TO expMAIN;
		new_name : STRING[EXPL_ITEM_LENGTH];
		size : STRING[15];
		side : BOOL;
	END_VAR
	VAR
		idx : DINT;
		idy : DINT;
		lSort : DINT;
	END_VAR
END_FUNCTION

FUNCTION WorkingStatus : USINT
	VAR_INPUT
		EXPL : REFERENCE TO expMAIN;
		str : UDINT;
		animation : USINT;
	END_VAR
END_FUNCTION

FUNCTION CreateCompletePath : BOOL
	VAR_INPUT
		path : STRING[EXPL_DIR_PATH_LENGTH];
		target : STRING[EXPL_ITEM_LENGTH];
		return_path : UDINT;
	END_VAR
	VAR
		tmp : STRING[EXPL_ITEM_LENGTH];
	END_VAR
END_FUNCTION

FUNCTION String2DataProvider : BOOL
	VAR_INPUT
		SourceString : UDINT;
		TargetString : UDINT;
	END_VAR
END_FUNCTION
```

#### LocalFunctions.st
```iecst
//******************************************************************************************************
// Create mappView data provider string
//******************************************************************************************************
FUNCTION String2DataProvider
	brsstrcpy(TargetString, ADR('{"value":"'));
	brsstrcat(TargetString, SourceString);
	brsstrcat(TargetString, ADR('","text":"'));
	brsstrcat(TargetString, SourceString);
	brsstrcat(TargetString, ADR('"}'));
	String2DataProvider := TRUE;
END_FUNCTION

//******************************************************************************************************
// Raise error function
//******************************************************************************************************
FUNCTION CreateError
	// Generate for known errors
	IF (nr = fiERR_NOT_ENOUGH_FREEMEM) THEN
		EXPL.ERR.text := 'not enough memory available on the target device';
	ELSIF (nr = fiERR_FILE_DEVICE) THEN
		EXPL.ERR.text := 'device is not connected';
	ELSIF (nr = fiERR_INVALID_PATH) THEN
		EXPL.ERR.text := 'directory is too long, does not exist or has invalid characters';
	ELSIF (nr = fiERR_DIR_NOT_EXIST) THEN
		EXPL.ERR.text := 'directory does not exist';
	ELSIF (nr = fiERR_FILE_DEVICE) THEN
		EXPL.ERR.text := 'directory path does not exist';
	ELSIF (nr = fiERR_DIR_ALREADY_EXIST) THEN
		EXPL.ERR.text := 'directory or file already exists';
	ELSIF (nr = fiERR_EXIST) THEN
		EXPL.ERR.text := 'error uploading file already exists';
	ELSE
		EXPL.ERR.text := text;
	END_IF
	// Convert to error structure
	IF (side = 0) THEN
		brsstrcat(ADR(EXPL.ERR.text), ADR(' on side a'));
	ELSE
		brsstrcat(ADR(EXPL.ERR.text), ADR(' on side b'));
	END_IF
	EXPL.ERR.no   	:= nr;
	EXPL.ERR.state 	:= step;
	// Set next step
	IF (step = EXP_READ_DIR_2) THEN
		CreateError := EXP_READ_DIR_3;
	ELSIF(step = EXP_FILE_UPLOAD_2) THEN
		CreateError := EXP_FILE_UPLOAD_3;
	ELSE
		// Reset all commands
		brsmemset(ADR(EXPL.CMD[side]), 0, SIZEOF(EXPL.CMD[side]));
		brsmemset(ADR(EXPL.CMD[NOT side]), 0, SIZEOF(EXPL.CMD[NOT side]));
		CreateError := EXP_WAIT;
	END_IF
END_FUNCTION

//******************************************************************************************************
// Create complete path string
//******************************************************************************************************
FUNCTION CreateCompletePath
	brsmemset(ADR(tmp), 0, EXPL_ITEM_LENGTH);
	brsstrcpy(return_path, ADR(path));

	// ------------------------------------------------------------------------------------------------
	// Filter directory name
	IF(brsmemcmp(ADR(target), ADR('(DIR)'), 5) = 0) THEN
		brsmemcpy(ADR(tmp), ADR(target)+5, brsstrlen(ADR(target))-5);
	ELSE
		brsstrcpy(ADR(tmp), ADR(target));
	END_IF

	// ------------------------------------------------------------------------------------------------
	// Create directory path
	brsstrcat(return_path, ADR('/'));
	brsstrcat(return_path, ADR(tmp));

	CreateCompletePath := FALSE;
END_FUNCTION

//******************************************************************************************************
// Working status
//******************************************************************************************************
FUNCTION WorkingStatus
	animation := animation+1;

	IF (animation = 80) THEN
		animation := 0;
	END_IF

	brsmemset(ADR(EXPL.status), 0, SIZEOF(EXPL.status));
	brsstrcpy(ADR(EXPL.status), str);
	CASE(animation) OF
		0..19	: brsstrcat(ADR(EXPL.status), ADR('/'));
		20..39	: brsstrcat(ADR(EXPL.status), ADR('-'));
		40..59	: brsstrcat(ADR(EXPL.status), ADR('\'));
		60..79	: brsstrcat(ADR(EXPL.status), ADR('|'));
	END_CASE;
	WorkingStatus := animation;
END_FUNCTION

//******************************************************************************************************
// Fill new folder or directory name
//******************************************************************************************************
FUNCTION InsertRecName
	// Set up start values for iteration
	IF (EXPL.DAT[side].item_num <> 0) THEN
		idy := EXPL.DAT[side].item_num - 1;
	END_IF
	idx := idy;

	// Start iteration	search
	WHILE (idy > 1) DO
		// Check current entry
		lSort := brsstrcmp(ADR(new_name), ADR(EXPL.DAT[side].item_list[idy]));
		// Solve new search range
		IF (idy MOD 2 = 0) THEN
			idy := idy / 2;
		ELSE
			idy := idy / 2 + 1;
		END_IF
		// New range is lower or higher than current
		IF (lSort > 0) THEN
			idx := idx + idy;
			IF (idx > UINT_TO_INT(EXPL.DAT[side].item_num)) THEN
				idx := EXPL.DAT[side].item_num;
			END_IF
		ELSE
			idx := idx - idy;
			IF (idx < 1) THEN
				idx := 1;
			END_IF
		END_IF
	END_WHILE;

	// New entry is this, next or previous
	lSort := brsstrcmp(ADR(new_name), ADR(EXPL.DAT[side].item_list[idx]));
	IF (lSort > 0 AND idx <> UINT_TO_INT(EXPL.DAT[side].item_num)) THEN
		idx := idx +1;
	ELSIF (idx > 0) THEN
		lSort := brsstrcmp(ADR(new_name), ADR(EXPL.DAT[side].item_list[idx-1]));
		IF (lSort < 0) THEN
			idx := idx - 1;
		END_IF
	END_IF

	// Force ".." at beginning of list
	IF (idx = 0 AND EXPL.DAT[side].item_list[0] = '..') THEN
		idx := idx + 1;
	END_IF
	// Move all data entrys backwards and fill in new entry
	IF(idx < EXPL_LIST_NUM) THEN
		brsmemmove(ADR(EXPL.DAT[side].item_list[idx+1]),ADR(EXPL.DAT[side].item_list[idx]), (EXPL.DAT[side].item_num - idx) * SIZEOF(EXPL.DAT[side].item_list[0]));
		brsmemmove(ADR(EXPL.DAT[side].item_size[idx+1]),ADR(EXPL.DAT[side].item_size[idx]), (EXPL.DAT[side].item_num - idx) * SIZEOF(EXPL.DAT[side].item_size[0]));
	END_IF
	brsstrcpy(ADR(EXPL.DAT[side].item_list[idx]), ADR(new_name));
	// Create data structure for vis size list
	brsstrcpy(ADR(EXPL.DAT[side].item_size[idx]), ADR(size));

	InsertRecName := TRUE;
END_FUNCTION

//******************************************************************************************************
// Is second string in first string
//******************************************************************************************************
FUNCTION IsInstr
	IF (brsstrlen(string1) > brsstrlen(string2)) THEN
		FOR idx:=0 TO brsstrlen(string1) - brsstrlen(string2) DO
			IF (brsmemcmp(string1 + idx, string2, brsstrlen(string2)) = 0) THEN
				IsInstr := TRUE;
				EXIT;
			END_IF
		END_FOR;
	END_IF
END_FUNCTION

//******************************************************************************************************
// Find second data in first data
//******************************************************************************************************
FUNCTION FindInMem
	IF (len1 > len2) THEN
		FOR idx:=0 TO len1 - len2 DO
			IF (brsmemcmp(data1 + idx, data2, len2) = 0) THEN
				FindInMem := idx;
				EXIT;
			END_IF
		END_FOR;
	END_IF
END_FUNCTION

//******************************************************************************************************
// Find and replace string
//******************************************************************************************************
FUNCTION ReplaceString
	IF (brsstrlen(dataSTR) > brsstrlen(searchSTR)) THEN
		FOR idx:=0 TO brsstrlen(dataSTR) - brsstrlen(searchSTR) DO
			IF (brsmemcmp(dataSTR + idx, searchSTR, brsstrlen(searchSTR)) = 0) THEN
				brsmemmove(dataSTR + idx + brsstrlen(replaceSTR), dataSTR + idx + brsstrlen(searchSTR), brsstrlen(dataSTR) - idx - brsstrlen(searchSTR));
				brsmemcpy(dataSTR + idx, replaceSTR, brsstrlen(replaceSTR));
				ReplaceString := TRUE;
				EXIT;
			END_IF
		END_FOR;
	END_IF
END_FUNCTION
```

### UsbGlobal.typ
```iecst
TYPE
	usbSTATE :
		(
		USB_WAIT, (*Wait for starting the Function chain*)
		USB_CREATE_NODE_ID_LIST, (*Create a list of Node-IDs from all active USB devices*)
		USB_READ_DEVICE_DATA, (*Read out the specific data from the Node-IDs*)
		USB_CHECK_DEVICE, (*Check file device data*)
		USB_LINK_DEVICE, (*Link file device*)
		USB_UNLINK_DEVICE, (*Unlink the File Device from specific path*)
		USB_ERROR (*Jump to this step in every case of Error occuring in the Function chain*)
		);
	usbCMD : 	STRUCT
		auto_scan : BOOL := TRUE; (*Scan USB ports automatically*)
		error_reset : BOOL; (*Reset error*)
	END_STRUCT;
	usbPAR : 	STRUCT
		state_machine : usbSTATE; (*State machine*)
		ignore_dongle : BOOL := TRUE; (*Ignoe B&R license dongle*)
		refresh_interval : UINT := 300; (*Intervall timer for USB device refresh*)
		is_connected : BOOL; (*Shows if a USB stick is connected*)
	END_STRUCT;
	usbERR : 	STRUCT
		no : UINT; (*Error number*)
		state : usbSTATE;
		text : STRING[80]; (*Error text*)
		active : BOOL;
	END_STRUCT;
	usbMAIN : 	STRUCT
		CMD : usbCMD; (*Command structure*)
		PAR : usbPAR; (*Parameter structure*)
		ERR : usbERR; (*Error structure*)
	END_STRUCT;
END_TYPE
```

### UsbGlobal.var
```iecst
VAR
	USB : usbMAIN;
END_VAR
```

### Program Logical/USBdevice/UsbDevice (IEC) - Sample for all AsUSB-Library-Functions

#### USBdevice.st - Cyclic code
```iecst
PROGRAM _INIT
END_PROGRAM

PROGRAM _CYCLIC

	CASE USB.PAR.state_machine OF
		// -----------------------------------------------------------------------------------------------------------
		// Wait state
		// -----------------------------------------------------------------------------------------------------------
		USB_WAIT:
			// Refresh USB data every X seconds when enabled
			IF USB.CMD.auto_scan = TRUE THEN
				TON_10ms_01(IN:=1, PT:=USB.PAR.refresh_interval);
				// Get new USB data
				IF(TON_10ms_01.Q) THEN
					TON_10ms_01(IN:=0);
					node := 0;
					brsmemset(ADR(usb_data), 0, SIZEOF(usb_data));
					USB.PAR.state_machine := USB_CREATE_NODE_ID_LIST;
				END_IF
			ELSE
				TON_10ms_01(IN:=0);
			END_IF;
			// Refresh USB data every X seconds when enabled
			IF USB.CMD.error_reset = TRUE THEN
				USB.PAR.state_machine := USB_ERROR;
			END_IF;
		// -----------------------------------------------------------------------------------------------------------
		// Get USB device list
		// -----------------------------------------------------------------------------------------------------------
		USB_CREATE_NODE_ID_LIST:
			UsbNodeListGet_0.enable := 1;
			UsbNodeListGet_0.pBuffer := ADR(node_id_buffer);
			UsbNodeListGet_0.bufferSize := SIZEOF(node_id_buffer);
			UsbNodeListGet_0.filterInterfaceClass := asusb_CLASS_MASS_STORAGE;
			UsbNodeListGet_0.filterInterfaceSubClass := 0;
			UsbNodeListGet_0;

			// --------------------------------------------------------------------------------------------------------------------
			// Success
			IF UsbNodeListGet_0.status = 0 THEN
				USB.PAR.state_machine := USB_READ_DEVICE_DATA;
				// No USB devices found
			ELSIF UsbNodeListGet_0.status = asusbERR_USB_NOTFOUND THEN
				// Unlink old device if it is gone now otherwise wait for next round
				IF(USB.PAR.is_connected) THEN
					USB.PAR.state_machine := USB_UNLINK_DEVICE;
				ELSE
					USB.PAR.state_machine := USB_WAIT;
				END_IF
				// Error
			ELSIF UsbNodeListGet_0.status <> ERR_FUB_BUSY THEN
				USB.ERR.state := USB.PAR.state_machine;
				USB.ERR.no := UsbNodeListGet_0.status;
				USB.ERR.text := 'error getting device list';
				USB.PAR.state_machine := USB_ERROR;
			END_IF;
		// -----------------------------------------------------------------------------------------------------------
		// Get device information
		// -----------------------------------------------------------------------------------------------------------
		USB_READ_DEVICE_DATA:
			UsbNodeGet_0.enable := 1;
			UsbNodeGet_0.nodeId := node_id_buffer[node];
			UsbNodeGet_0.pBuffer := ADR(usb_data[node]);
			UsbNodeGet_0.bufferSize := SIZEOF (usb_data[node]);
			UsbNodeGet_0;

			// --------------------------------------------------------------------------------------------------------------------
			// Success
			IF UsbNodeGet_0.status = 0 THEN
				// Make sure we have enough space to store USB data, proceed with next USB.PAR.state_machine when all devices are detetced
				IF (node = UsbNodeListGet_0.listNodes - 1) OR (node > SIZEOF(usb_data)/SIZEOF(usb_data[0])) THEN
					idx := 0;
					USB.PAR.state_machine := USB_CHECK_DEVICE;
					// Get next USB device
				ELSE
					node := node + 1;
				END_IF;
				// Error
			ELSIF UsbNodeGet_0.status <> ERR_FUB_BUSY THEN
				USB.ERR.state := USB.PAR.state_machine;
				USB.ERR.no := UsbNodeGet_0.status;
				USB.ERR.text := 'error getting device data';
				USB.PAR.state_machine := USB_ERROR;
			END_IF;
		// -----------------------------------------------------------------------------------------------------------
		// Check if device is connected
		// -----------------------------------------------------------------------------------------------------------
		USB_CHECK_DEVICE:
			// Check if device is already linked
			IF(USB.PAR.is_connected) THEN
				// Device is already linked, return to wait state
				IF(brsmemcmp(ADR(usb_data_linked), ADR(usb_data[idx]), SIZEOF(usb_data[idx])) = 0) THEN
					USB.PAR.state_machine := USB_WAIT;
					// Check next device
				ELSIF(idx < node) THEN
					idx := idx + 1;
					// Unlink device if it is gone
				ELSE
					USB.PAR.state_machine := USB_UNLINK_DEVICE;
				END_IF
			ELSE
				// Check if B&R dongle should be excluded from list
				IF(USB.PAR.ignore_dongle=TRUE AND usb_data[idx].productId=1001 AND usb_data[idx].vendorId=1615) THEN
					IF(idx < node) THEN
						idx := idx + 1;
					ELSE
						USB.PAR.state_machine := USB_WAIT;
					END_IF
				ELSE
					USB.PAR.state_machine := USB_LINK_DEVICE;
				END_IF
			END_IF
		// -----------------------------------------------------------------------------------------------------------
		// Link device
		// -----------------------------------------------------------------------------------------------------------
		USB_LINK_DEVICE:
			// Create device string
			brsstrcpy(ADR(device_param), ADR('/DEVICE='));
			brsstrcat(ADR(device_param), ADR(usb_data[node].ifName));
			// Link device
			DevLink_0.enable := 1;
			DevLink_0.pDevice := ADR('USB_DEVICE');
			DevLink_0.pParam := ADR(device_param);
			DevLink_0;

			// --------------------------------------------------------------------------------------------------------------------
			// Success
			IF DevLink_0.status = 0 THEN
				brsmemcpy(ADR(usb_data_linked), ADR(usb_data[node]), SIZEOF(usb_data[node]));
				USB.PAR.is_connected := TRUE;
				USB.PAR.state_machine := USB_WAIT;
				// Error
			ELSIF DevLink_0.status <> ERR_FUB_BUSY THEN
				USB.ERR.state := USB.PAR.state_machine;
				USB.ERR.no := DevLink_0.status;
				USB.ERR.text := 'error linking device';
				USB.PAR.state_machine := USB_ERROR;
			END_IF;
		// -----------------------------------------------------------------------------------------------------------
		// UnLink device
		// -----------------------------------------------------------------------------------------------------------
		USB_UNLINK_DEVICE:
			DevUnlink_0.enable := 1;
			DevUnlink_0.handle := DevLink_0.handle;
			DevUnlink_0;

			// --------------------------------------------------------------------------------------------------------------------
			// Success
			IF DevUnlink_0.status = 0 THEN
				brsmemset(ADR(usb_data_linked), 0, SIZEOF(usb_data_linked));
				USB.PAR.is_connected := FALSE;
				IF(UsbNodeListGet_0.status = asusbERR_USB_NOTFOUND) THEN
					USB.PAR.state_machine := USB_WAIT;
				ELSE
					idx := 0;
					USB.PAR.state_machine := USB_CHECK_DEVICE;
				END_IF
				// Error
			ELSIF DevUnlink_0.status <> ERR_FUB_BUSY THEN
				USB.ERR.state := USB.PAR.state_machine;
				USB.ERR.no := DevUnlink_0.status;
				USB.ERR.text := 'error unlinking device';
				USB.PAR.state_machine := USB_ERROR;
			END_IF;
		// -----------------------------------------------------------------------------------------------------------
		// Error state
		// -----------------------------------------------------------------------------------------------------------
		USB_ERROR:
			// Get more error information
			IF(USB.ERR.no = 0) THEN
				USB.ERR.no := FileIoGetSysError();
			END_IF
			USB.ERR.active := TRUE;
			USB.PAR.is_connected := FALSE;

			// Unlink device
			DevUnlink_0.enable := 1;
			DevUnlink_0.handle := DevLink_0.handle;
			DevUnlink_0;

			// Reset error
			IF(USB.CMD.error_reset AND DevUnlink_0.status <> ERR_FUB_BUSY) THEN
				USB.CMD.error_reset := FALSE;
				USB.ERR.active := FALSE;
				USB.ERR.no := 0;
				brsmemset(ADR(USB.ERR.text), 0, SIZEOF(USB.ERR.text));
				USB.PAR.state_machine := USB_WAIT;
			END_IF
	END_CASE;

END_PROGRAM

PROGRAM _EXIT
	REPEAT
		DevUnlink_0.enable := 1;
		DevUnlink_0.handle := DevLink_0.handle;
		DevUnlink_0;
		UNTIL DevUnlink_0.status <> ERR_FUB_BUSY
	END_REPEAT;
END_PROGRAM
```

#### USBdevice.var - Data for read_data Task
```iecst
(*----------------------------------------------------------------------------------------------------------------------------------------------------------------------------------------------------------------------------------------------------------------------*)
(*Local functions*)
VAR
	TON_10ms_01 : TON_10ms;
	UsbNodeListGet_0 : UsbNodeListGet; (*Type of FUB UsbNodeListGet*)
	UsbNodeGet_0 : UsbNodeGet; (*Type of FUB UsbNodeGet*)
	DevLink_0 : DevLink; (*Type of FUB DevLink*)
	DevUnlink_0 : DevUnlink; (*Type of FUB DevUnlink*)
END_VAR
(*----------------------------------------------------------------------------------------------------------------------------------------------------------------------------------------------------------------------------------------------------------------------*)
(*Local variables*)
VAR
	device_param : STRING[80]; (*Connection path of USB device*)
	usb_data : ARRAY[0..4] OF usbNode_typ; (*Data of all available USB devices*)
	usb_data_linked : usbNode_typ; (*Data of the linked device*)
	node_id_buffer : ARRAY[0..4] OF UDINT; (*Different nodeIDs saved in array-elements*)
	node : USINT; (*Node number*)
	idx : USINT;
END_VAR
```

### NetGlobal.typ
```iecst
TYPE
	netSTATE :
		(
		NET_WAIT, (*Function step: Wait for starting the Function chain*)
		NET_LINK_DEVICE, (*Function step: Link file device*)
		NET_UNLINK_DEVICE, (*Function step: Unlink the File Device from specific path*)
		NET_ERROR (*Function step: Jump to this step in every case of Error occuring in the Function chain*)
		);
	netCMD : 	STRUCT
		connect : BOOL := TRUE; (*Connect to network share*)
		error_reset : BOOL; (*Reset error*)
	END_STRUCT;
	netPAR : 	STRUCT
		state_machine : netSTATE; (*State machine*)
		server_name : STRING[80]; (*Use server name*)
		server_ip : STRING[80] := '192.168.0.10'; (*or IP address*)
		server_port : STRING[80]; (*Uses default port when empty*)
		server_protocol : STRING[80] := 'ftp'; (*Type of network connection*)
		server_domain : STRING[80]; (*Domain name*)
		server_share : STRING[80] := 'share'; (*Name of the shared folder*)
		user_name : STRING[80] := 'user'; (*User name*)
		user_password : STRING[80] := 'password'; (*User password*)
		enable_connect : BOOL; (*Enable button connect*)
		is_linked : BOOL; (*Network share is connected*)
	END_STRUCT;
	netERR : 	STRUCT
		no : UINT; (*Error number*)
		state : netSTATE;
		text : STRING[80]; (*Error text*)
		active : BOOL;
	END_STRUCT;
	netMAIN : 	STRUCT
		CMD : netCMD; (*Command structure*)
		PAR : netPAR; (*Parameter structure*)
		ERR : netERR; (*Error structure*)
	END_STRUCT;
END_TYPE
```

### NetGlobal.var
```iecst
VAR
	NET : netMAIN;
END_VAR
```

### Program Logical/NETdevice/NetDevice (IEC)

#### Main.st - Init, cyclic, exit code
```iecst
PROGRAM _INIT
	(* Insert code here *)

END_PROGRAM

PROGRAM _CYCLIC

	CASE NET.PAR.state_machine OF
		// -----------------------------------------------------------------------------------------------------------
		// Wait state
		// -----------------------------------------------------------------------------------------------------------
		NET_WAIT:
			NET.PAR.enable_connect := TRUE;
			// --------------------------------------------------------------------------------------------------------------------
			// Connect to server
			IF(NET.CMD.connect) THEN
				IF(NET.PAR.is_linked) THEN
					DevUnlink_0.enable := 0;
					DevUnlink_0;
					IF (DevUnlink_0.status = ERR_FUB_ENABLE_FALSE) THEN
						NET.PAR.state_machine := NET_UNLINK_DEVICE;
					END_IF
				ELSE
					DevLink_0.enable := 0;
					DevLink_0;
					IF (DevLink_0.status = ERR_FUB_ENABLE_FALSE) THEN
						NET.PAR.state_machine := NET_LINK_DEVICE;
					END_IF
				END_IF
			END_IF
			// --------------------------------------------------------------------------------------------------------------------
			// Disconnect from server
			IF(NET.CMD.error_reset) THEN
				IF(NET.PAR.is_linked) THEN
					DevUnlink_0.enable := 0;
					DevUnlink_0;
					NET.PAR.state_machine := NET_UNLINK_DEVICE;
				ELSE
					NET.CMD.error_reset := FALSE;
				END_IF
			END_IF
		// -----------------------------------------------------------------------------------------------------------
		// Link device
		// -----------------------------------------------------------------------------------------------------------
		NET_LINK_DEVICE:
			// Create device string
			NET.PAR.enable_connect := FALSE;
			brsmemset(ADR(device_param), 0, SIZEOF(device_param));
			IF(brsstrcmp(ADR(NET.PAR.server_name), ADR('')) <> 0) THEN
				brsstrcat(ADR(device_param), ADR('/SNAME='));
				brsstrcat(ADR(device_param), ADR(NET.PAR.server_name));
				brsstrcat(ADR(device_param), ADR(' '));
			END_IF
			IF(brsstrcmp(ADR(NET.PAR.server_ip), ADR('')) <> 0) THEN
				brsstrcat(ADR(device_param), ADR('/SIP='));
				brsstrcat(ADR(device_param), ADR(NET.PAR.server_ip));
				brsstrcat(ADR(device_param), ADR(' '));
			END_IF
			IF(brsstrcmp(ADR(NET.PAR.server_protocol), ADR('')) <> 0) THEN
				brsstrcat(ADR(device_param), ADR('/PROTOCOL='));
				brsstrcat(ADR(device_param), ADR(NET.PAR.server_protocol));
				brsstrcat(ADR(device_param), ADR(' '));
			END_IF
			IF(brsstrcmp(ADR(NET.PAR.server_port), ADR('')) <> 0) THEN
				brsstrcat(ADR(device_param), ADR('/PORT='));
				brsstrcat(ADR(device_param), ADR(NET.PAR.server_port));
				brsstrcat(ADR(device_param), ADR(' '));
			END_IF
			IF(brsstrcmp(ADR(NET.PAR.server_domain), ADR('')) <> 0) THEN
				brsstrcat(ADR(device_param), ADR('/DOMAIN='));
				brsstrcat(ADR(device_param), ADR(NET.PAR.server_domain));
				brsstrcat(ADR(device_param), ADR(' '));
			END_IF
			IF(brsstrcmp(ADR(NET.PAR.server_share), ADR('')) <> 0) THEN
				brsstrcat(ADR(device_param), ADR('/SHARE='));
				brsstrcat(ADR(device_param), ADR(NET.PAR.server_share));
				brsstrcat(ADR(device_param), ADR(' '));
			END_IF
			IF(brsstrcmp(ADR(NET.PAR.user_name), ADR('')) <> 0) THEN
				brsstrcat(ADR(device_param), ADR('/USER='));
				brsstrcat(ADR(device_param), ADR(NET.PAR.user_name));
				brsstrcat(ADR(device_param), ADR(' '));
			END_IF
			IF(brsstrcmp(ADR(NET.PAR.user_password), ADR('')) <> 0) THEN
				brsstrcat(ADR(device_param), ADR('/PASSWORD='));
				brsstrcat(ADR(device_param), ADR(NET.PAR.user_password));
				brsstrcat(ADR(device_param), ADR(' '));
			END_IF

			// Link device
			DevLink_0.enable := 1;
			DevLink_0.pDevice := ADR('NET_DEVICE');
			DevLink_0.pParam := ADR(device_param);
			DevLink_0;

			// --------------------------------------------------------------------------------------------------------------------
			// Success
			IF DevLink_0.status = 0 THEN
				device_handle := DevLink_0.handle;
				NET.PAR.is_linked := TRUE;
				NET.CMD.connect := FALSE;
				NET.PAR.state_machine := NET_WAIT;
			// --------------------------------------------------------------------------------------------------------------------
			// Abort command
			ELSIF(NET.CMD.error_reset) THEN
				NET.CMD.error_reset := FALSE;
				NET.CMD.connect := FALSE;
				NET.PAR.state_machine := NET_WAIT;
				// Error
			ELSIF DevLink_0.status <> ERR_FUB_BUSY THEN
				NET.ERR.state := NET.PAR.state_machine;
				NET.ERR.no := DevLink_0.status;
				NET.ERR.text := 'error linking device';
				NET.PAR.state_machine := NET_ERROR;
			END_IF;
		// -----------------------------------------------------------------------------------------------------------
		// UnLink device
		// -----------------------------------------------------------------------------------------------------------
		NET_UNLINK_DEVICE:
			NET.PAR.enable_connect := FALSE;
			DevUnlink_0.enable := 1;
			DevUnlink_0.handle := device_handle;
			DevUnlink_0;

			// --------------------------------------------------------------------------------------------------------------------
			// Success
			IF DevUnlink_0.status = 0 THEN
				NET.PAR.is_linked := FALSE;
				IF(NET.CMD.connect) THEN
					DevLink_0.enable := 0;
					DevLink_0;
					NET.PAR.state_machine := NET_LINK_DEVICE;
				ELSE
					NET.CMD.error_reset := FALSE;
					NET.PAR.state_machine := NET_WAIT;
				END_IF
			// Error
			ELSIF DevUnlink_0.status <> ERR_FUB_BUSY THEN
				NET.CMD.error_reset := FALSE;
				NET.ERR.state := NET.PAR.state_machine;
				NET.ERR.no := DevUnlink_0.status;
				NET.ERR.text := 'error unlinking device';
				NET.PAR.state_machine := NET_ERROR;
			END_IF;
		// -----------------------------------------------------------------------------------------------------------
		// Error step
		// -----------------------------------------------------------------------------------------------------------
		NET_ERROR:
			// Reset commands
			NET.PAR.enable_connect := FALSE;
			NET.CMD.connect := FALSE;

			// Get more error information
			IF(NET.ERR.no = 0) THEN
				NET.ERR.no := FileIoGetSysError();
			END_IF
			NET.ERR.active := TRUE;
			IF(NET.ERR.no=26228) THEN
				brsstrcpy(ADR(NET.ERR.text), ADR('connection rejected: check network protocol, username and password'));
			ELSIF(DevLink_0.status = fiERR_DEVICE_ALREADY_EXIST) THEN
				brsstrcpy(ADR(NET.ERR.text), ADR('device is already connected'));
			END_IF

			// Reset error
			IF(NET.CMD.error_reset) THEN
				NET.CMD.error_reset := FALSE;
				NET.ERR.active := FALSE;
				NET.ERR.no := 0;
				brsmemset(ADR(NET.ERR.text), 0, SIZEOF(NET.ERR.text));
				NET.PAR.state_machine := NET_WAIT;
			END_IF
	END_CASE;

END_PROGRAM

PROGRAM _EXIT
	REPEAT
		DevUnlink_0.enable := 1;
		DevUnlink_0.handle := DevLink_0.handle;
		DevUnlink_0;
		UNTIL DevUnlink_0.status <> ERR_FUB_BUSY
	END_REPEAT;
END_PROGRAM
```

#### Variables.var - Local variables
```iecst
(*----------------------------------------------------------------------------------------------------------------------------------------------------------------------------------------------------------------------------------------------------------------------*)
(*Local functions*)
VAR
	DevLink_0 : DevLink; (*Type of FUB DevLink*)
	DevUnlink_0 : DevUnlink; (*Type of FUB DevUnlink*)
END_VAR
(*----------------------------------------------------------------------------------------------------------------------------------------------------------------------------------------------------------------------------------------------------------------------*)
(*Local variables*)
VAR
	device_param : STRING[200]; (*Connection path of USB device*)
	device_handle : UDINT;
END_VAR
```

### DatumCasGlobal.var
```iecst
VAR
	PLC_Cas : PLC_Cas_typ;
	PLC_Datum : PLC_Datum_typ;
	Sekunda_STR : STRING[2];
	Minuta_STR : STRING[2];
	Hodina_STR : STRING[2];
	Den_STR : STRING[2];
	Mesiac_STR : STRING[2];
	Rok_STR_4_Znaky : STRING[4];
	Rok_STR_2_Znaky : STRING[2];
END_VAR
```

### DatumCasGlobal.typ
```iecst
TYPE
	PLC_Cas_typ : 	STRUCT
		Sekundy : USINT;
		Minuty : USINT;
		Hodiny : USINT;
	END_STRUCT;
	PLC_Datum_typ : 	STRUCT
		Den : USINT;
		Mesiac : USINT;
		Rok : UINT;
	END_STRUCT;
END_TYPE
```

### Program Logical/DatumCasPLC/DatumCasPLC (IEC)

#### Main.st - Init, cyclic, exit code
```iecst
PROGRAM _INIT
	(* Insert code here *)

END_PROGRAM

PROGRAM _CYCLIC

	//Vyčítavanie systémového času//
	DTGetTime_1.enable:= TRUE;
	DTGetTime_1();
	DT_TO_DTStructure(DTGetTime_1.DT1,ADR(PLC_DatumCas));

	PLC_Cas.Sekundy:= PLC_DatumCas.second;
	PLC_Cas.Minuty:= PLC_DatumCas.minute;
	PLC_Cas.Hodiny:= PLC_DatumCas.hour;

	PLC_Datum.Den:= PLC_DatumCas.day;
	PLC_Datum.Mesiac:= PLC_DatumCas.month;
	PLC_Datum.Rok:= PLC_DatumCas.year;

	//Prevod času na String//
	//Sekundy//
	IF PLC_Cas.Sekundy < 10 THEN
		Sekundy_String:= USINT_TO_STRING(PLC_Cas.Sekundy);
		Sekunda_STR:= '0';
		brsstrcat(ADR(Sekunda_STR),ADR(Sekundy_String));
	ELSE
		Sekunda_STR:= USINT_TO_STRING(PLC_Cas.Sekundy);
	END_IF

	//Minuty//
	IF PLC_Cas.Minuty < 10 THEN
		Minuty_String:= USINT_TO_STRING(PLC_Cas.Minuty);
		Minuta_STR:= '0';
		brsstrcat(ADR(Minuta_STR),ADR(Minuty_String));
	ELSE
		Minuta_STR:= USINT_TO_STRING(PLC_Cas.Minuty);
	END_IF

	//Hodiny//
	IF PLC_Cas.Hodiny < 10 THEN
		Hodiny_String:= USINT_TO_STRING(PLC_Cas.Hodiny);
		Hodina_STR:= '0';
		brsstrcat(ADR(Hodina_STR),ADR(Hodiny_String));
	ELSE
		Hodina_STR:= USINT_TO_STRING(PLC_Cas.Hodiny);
	END_IF

	//Prevod dátumu na String//
	//Deň//
	IF PLC_Datum.Den < 10 THEN
		Den_String:= USINT_TO_STRING(PLC_Datum.Den);
		Den_STR:= '0';
		brsstrcat(ADR(Den_STR),ADR(Den_String));
	ELSE
		Den_STR:= USINT_TO_STRING(PLC_Datum.Den);
	END_IF

	//Masiac//
	IF PLC_Datum.Mesiac < 10 THEN
		Mesiac_String:= USINT_TO_STRING(PLC_Datum.Mesiac);
		Mesiac_STR:= '0';
		brsstrcat(ADR(Mesiac_STR),ADR(Mesiac_String));
	ELSE
		Mesiac_STR:= USINT_TO_STRING(PLC_Datum.Mesiac);
	END_IF

	//Rok - 4 znaky//
	Rok_STR_4_Znaky:= UINT_TO_STRING(PLC_Datum.Rok);

	//Rok - posledné 2 znaky//
	length := brsstrlen(ADR(Rok_STR_4_Znaky)); //Zistí počet znakov//

	IF length >= 4 THEN
		brsmemcpy(ADR(PoleUSINT),ADR(Rok_STR_4_Znaky),SIZEOF(Rok_STR_4_Znaky));
		i := PoleUSINT[length-2]; //Vyčítanie predposledného znaku//
		brsstrcpy(ADR(DvaZnaky),ADR(i));
		i := PoleUSINT[length-1]; //Vyčítanie posledneho znaku//
		brsstrcat(ADR(DvaZnaky),ADR(i));
	END_IF

	Rok_STR_2_Znaky:= DvaZnaky;

END_PROGRAM

PROGRAM _EXIT
	(* Insert code here *)

END_PROGRAM
```

#### Variables.var - Local variables
```iecst
VAR
	PLC_DatumCas : DTStructure;
	DTGetTime_1 : DTGetTime;
	Sekundy_String : STRING[2];
	Minuty_String : STRING[2];
	Hodiny_String : STRING[2];
	Den_String : STRING[2];
	Mesiac_String : STRING[2];
	length : UDINT;
	PoleUSINT : ARRAY[0..3] OF USINT;
	i : USINT;
	DvaZnaky : STRING[2];
END_VAR
```

### Poznamky.txt
```
Prihlasovacie údaje na FTP:
Login - admin
Heslo - vlmardo

Prihlasovacie údaje do Safety:
Heslo - vlmardo

//*********APC Windows*************//
Heslo - vlmardoDMP

//**********Vzdialená plocha**********//
192.168.122.3
Meno - remote
Heslo - vlmardo

//***********Prístup na FTP SSD disk PLC*******//
IP 192.168.122.3
Meno - remote
Heslo - vlmardo

//************Prístup na FTP kameru č.1 na disku PLC*********//
IP 192.168.122.4
Meno - cam1
Heslo - .cam1

//************Prístup na FTP Panasonic*******************//
IP 192.168.100.164
Meno - designMP
Heslo - Ftp4PAN2020

Pre spojenie je potrebné vypnúť wifi

**********Pracovisko 1*************
Výťah:
- Servo zdvihu výťahu - prevod 5mm/ot
Šrobovanie:
- Servo manipulatora Os X - prevod 10mm/ot
- Servo manipulatora Os Y - prevod 10mm/ot

***********Pracovisko 2*************
Zakladač izolácie:
- Servo zdvihu - prevod 10mm/ot  Celkový zdvih 100mm
- Servo pojazdu vozíka - prevod 132mm/ot
Šrobovanie:
- Servo manipulatora Os X - prevod 10mm/ot
- Servo manipulatora Os Y - prevod 10mm/ot
Zváranie:
- Servo zdvihu zvárania - prevod 10mm/ot Celkový zdvih 310mm

*****************Číslovanie kamier*************************
CAM 1 - Control Unit CAM 4
CAM 2 - Control Unit CAM 1
CAM 4 - Control Unit CAM 2
CAM 6 - Control Unit CAM 3
CAM 7 - Control Unit CAM 5
CAM 10 - Control Unit CAM 7
CAM 11 - Control Unit CAM 9
CAM 12 - Control Unit CAM 8
CAM 13 - Control Unit CAM 10
CAM 15 - Control Unit CAM 11
CAM 16 - Control Unit CAM 12
CAM 17 - Control Unit CAM 6

CAM 9 - Smart kamera CAM9
IP kamerového systému 192.168.122.128
Heslo - vision

**************************Postup kalibrácie vysunutia šróbovačiek***********************************
- na pracovisku zacentrujeme paletku

********P1 Skrutkovanie*************
Skrutkovačka K30 - dištanc 60mm  východzia poloha
                 - opretie o paletku  koncová poloha

Skrutkovačka M5 - dištanc 60mm východzia poloha
                - opretie o paletku koncová poloha

Skrutkovačka M4 - dištanc 60mm východzia poloha
                - dištanc 12mm koncová poloha

*******P2 Maticovačka***************
Skrutkovačka matice M4 - dištanc 52mm východzia poloha
                       - dištanc 12mm koncová poloha

*******P2 Skrutkovanie****************
Skrutkovačka M6 - dištanc 72mm východzia poloha
                - dištanc 15mm koncová poloha

Skrutkovačka M4 - dištanc 87mm východzia poloha
                - dištanc 27mm koncová poloha

Skrutkovačka M5 - dištanc 115 mm východzia poloha
                - max vysunutie skrutkovačky koncová poloha

*******P3 Skrutkovanie******************
Skrutkovačka K40 - dištanc 52,5mm východzia poloha
                 - opretie o paletku  koncová poloha

Skrutkovačka M5 - dištanc 60mm  východzia poloha
                - opretie o paletku  koncová poloha

*****************************************************Kalibračné hodnoty skrutkovačiek***********************************************************
/Model 5H/

Srutkovanie 1:
Lavá K30 - 44.6 až 44.9
Pravá K30 - 44.5 až 44.8
Lavá M5 - 31.3 až 31.7
Pravá M5 - 31.0 až 31.5
Stredná M5 - 31.4 až 31.8

Skrutkovanie matice:
Vysunutie skrutkovačky - 37.5 až 37.8

Skrutkovanie 2:
Lavá M5 - 40.7 až 41.1
Pravá M5 - 40.7 až 41.0
Stredná M4 - 15.8 až 16.3

Skrutkovanie 3:
Stredná M5 - 42.0 až 42.3
```
